(* CODESYS project LockSalve1_SC.export

Project tree, tasks and I/O mapping:
  function block LockSalve1_SC [ST]
*)

// LockSalve1_SC
FUNCTION_BLOCK LockSalve1_SC
VAR_INPUT
	EStop_IN:BOOL;                   //急停
	Forced_IN:BOOL;                  //强制
	ArmLimit_IN:BOOL;                //臂架限位
	LegOK_IN:BOOL;                   //支腿压实
	RTRotate_IN:SINT;
	ArmAngle_IN:SINT;
	ArmLength_IN:SINT;
END_VAR
VAR_OUTPUT
	StopValve_OUT:BOOL;                    //截止阀
	UnloadValve_OUT:BOOL;                  //卸荷阀
	Fault_OUT:BOOL;                        //互锁故障
END_VAR
VAR
	M1:BOOL;
	M2:BOOL;
	T1: TOF;
	T2: TON;
END_VAR

//有臂架检测和软退检测
IF RTRotate_IN=0 AND ArmAngle_IN=0 AND ArmLength_IN=0 THEN
	M1:=FALSE;
ELSE
	M1:=TRUE;
END_IF

T1(IN:=M1 , PT:=T#3S , Q=> , ET=> );
T2(IN:=Forced_IN , PT:=T#30S , Q=> , ET=> );
IF Forced_IN=TRUE AND T2.Q=FALSE THEN
	M2:=TRUE;
ELSE
	M2:=FALSE;
END_IF
IF EStop_IN=TRUE THEN
	IF ArmLimit_IN=TRUE OR M2=TRUE THEN
		StopValve_OUT:=FALSE;
	ELSE
		StopValve_OUT:=TRUE;
	END_IF
	IF LegOK_IN=TRUE OR M2=TRUE THEN
		IF T1.Q=FALSE THEN
			UnloadValve_OUT:=FALSE;
		ELSE
			UnloadValve_OUT:=TRUE;
		END_IF
	ELSE
		UnloadValve_OUT:=FALSE;
	END_IF
ELSE
	StopValve_OUT:=TRUE;
	UnloadValve_OUT:=FALSE;
END_IF

IF ArmLimit_IN=FALSE AND LegOK_IN=FALSE THEN
	Fault_OUT:=TRUE;
ELSE
	Fault_OUT:=FALSE;
END_IF

END_FUNCTION_BLOCK
